SUBAPPLICATION Servo_Slider_OPC (* Demo: Servo an Output_Q2, Winkel 0-180 Grad per Web-Slider (OPC-UA), aktueller Winkel wird als Echo zurueckpubliziert *)
  (* Standard: 61499-2; Description: Copyright (c) 2026 Meisterschulen am Ostbahnhof This program and the accompanying materials are made available under the terms of the Eclipse Public License 2.0 which is available at https://www.eclipse.org/legal/epl-2.0/ SPDX-License-Identifier: EPL-2.0 *)
  (* Version 1.0, 2026-10-05, Franz Höpfinger, Meisterschulen am Ostbahnhof, initial API and implementation and/or initial documentation *)
  PACKAGE Meins::Servo_Slider_OPC;
  IMPORT Meins::Servo_Slider_OPC::SubStrings::SERVO_Q2_ANGLE_SET;
  IMPORT Meins::Servo_Slider_OPC::SubStrings::SERVO_Q2_ANGLE;
  IMPORT logiBUS::io::DQ::logiBUS_DO::Output_Q2;
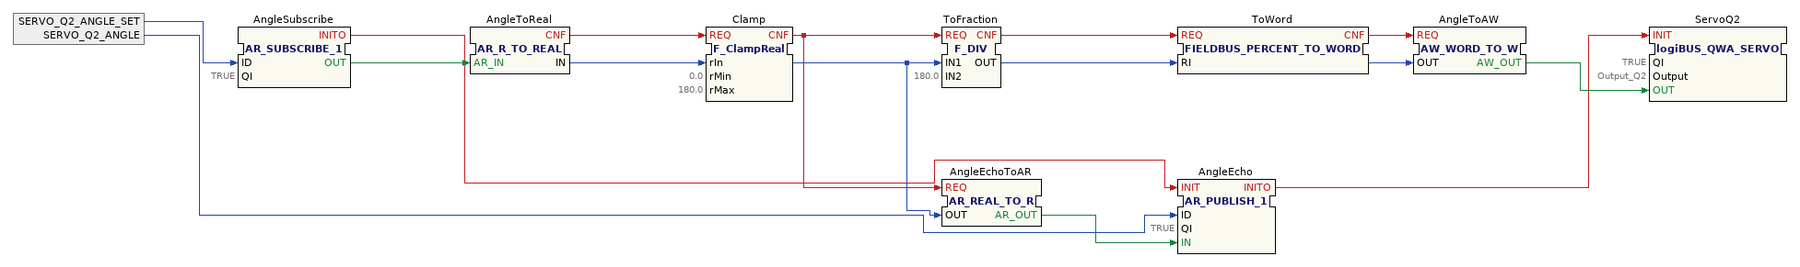
  FBS
    AngleSubscribe : adapter::net::AR_SUBSCRIBE_1(QI := TRUE);
    AngleToReal : adapter::conversion::unidirectional::AR_R_TO_REAL;
    Clamp : logiBUS::signalprocessing::clamp::F_ClampReal(rMin := 0.0, rMax := 180.0);
    ToFraction : iec61131::arithmetic::F_DIV(IN2 := 180.0);
    ToWord : eclipse4diac::signalprocessing::FIELDBUS_PERCENT_TO_WORD;
    AngleToAW : adapter::conversion::unidirectional::AW_WORD_TO_W;
    ServoQ2 : logiBUS::io::DO_SERVO::logiBUS_QWA_SERVO(QI := TRUE, Output := Output_Q2);
    AngleEchoToAR : adapter::conversion::unidirectional::AR_REAL_TO_R;
    AngleEcho : adapter::net::AR_PUBLISH_1(QI := TRUE);
  END_FBS
  EVENT_CONNECTIONS
    AngleToReal.CNF TO Clamp.REQ;
    Clamp.CNF TO ToFraction.REQ;
    Clamp.CNF TO AngleEchoToAR.REQ;
    ToFraction.CNF TO ToWord.REQ;
    ToWord.CNF TO AngleToAW.REQ;
    AngleSubscribe.INITO TO AngleEcho.INIT;
    AngleEcho.INITO TO ServoQ2.INIT;
  END_CONNECTIONS
  DATA_CONNECTIONS
    SERVO_Q2_ANGLE_SET TO AngleSubscribe.ID;
    SERVO_Q2_ANGLE TO AngleEcho.ID;
    AngleToReal.IN TO Clamp.rIn;
    Clamp. TO ToFraction.IN1;
    ToFraction.OUT TO ToWord.RI;
    ToWord. TO AngleToAW.OUT;
    Clamp. TO AngleEchoToAR.OUT;
  END_CONNECTIONS
  ADAPTER_CONNECTIONS
    AngleSubscribe.OUT TO AngleToReal.AR_IN;
    AngleToAW.AW_OUT TO ServoQ2.OUT;
    AngleEchoToAR.AR_OUT TO AngleEcho.IN;
  END_CONNECTIONS
END_SUBAPPLICATION
